ELSIF  parts.axes.statuses.initializationStatus.shutdown OR 
    parts.cover.statuses.initializationStatus.shutdown OR 
    parts.hydraulics.statuses.initializationStatus.shutdown OR 
    parts.m1.statuses.initializationStatus.shutdown OR 
    parts.m2.statuses.initializationStatus.shutdown OR 
    parts.m3.statuses.initializationStatus.shutdown OR 
    parts.safety.statuses.initializationStatus.shutdown OR 
    parts.services.statuses.initializationStatus.shutdown OR 
    parts.telemetry.statuses.initializationStatus.shutdown THEN

            statuses.initializationStatus(superState := TRUE, state := InitializationStates.SHUTDOWN);
ELSE
    statuses.initializationStatus(superState := FALSE);
END_IF


IF statuses.initializationStatus.initialized THEN
    IF statuses.healthStatus.bad THEN
        actualStatus := 'ERROR';
    ELSIF statuses.healthStatus.warning THEN
        actualStatus := 'Warning';
    ELSIF statuses.healthStatus.good THEN 
        IF statuses.busyStatus.busy THEN
            actualStatus := 'Busy';
        ELSIF statuses.busyStatus.idle THEN
            actualStatus := 'Idle';
        ELSE
            actualStatus := 'UNKNOWN';
        END_IF
    ELSE
        actualStatus := 'UNKNOWN';
	END_IF
ELSE
    actualStatus := InitializationStatusToString(statuses.initializationStatus);
END_IF


isInstrumentActive := parts.m3.statuses.busyStatus.idle AND parts.m3.actualKnownPositionID <> M3PositionIDs.UNKNOWN;

IF processes.changeInstrument.isBusy() THEN
    activeInstrumentName := 'Changing...';
    activeInstrumentNumber := -1;
ELSE
    IF isInstrumentActive THEN
        activeInstrumentName := parts.m3.actualKnownPositionName;
        
        IF activeInstrumentName = config.instruments.instrument0.name THEN
            activeInstrumentNumber := 0;
            activeInstrument := config.instruments.instrument0;
        ELSIF activeInstrumentName = config.instruments.instrument1.name THEN
            activeInstrumentNumber := 1;
            activeInstrument := config.instruments.instrument1;
        ELSIF activeInstrumentName = config.instruments.instrument2.name THEN
            activeInstrumentNumber := 2;
            activeInstrument := config.instruments.instrument2;
        ELSIF activeInstrumentName = config.instruments.instrument3.name THEN
            activeInstrumentNumber := 3;
            activeInstrument := config.instruments.instrument3;
        ELSIF activeInstrumentName = config.instruments.instrument4.name THEN
            activeInstrumentNumber := 4;
            activeInstrument := config.instruments.instrument4;
        ELSIF activeInstrumentName = config.instruments.instrument5.name THEN
            activeInstrumentNumber := 5;
            activeInstrument := config.instruments.instrument5;
        ELSIF activeInstrumentName = config.instruments.instrument6.name THEN
            activeInstrumentNumber := 6;
            activeInstrument := config.instruments.instrument6;
        ELSIF activeInstrumentName = config.instruments.instrument7.name THEN
            activeInstrumentNumber := 7;
            activeInstrument := config.instruments.instrument7;
        ELSIF activeInstrumentName = config.instruments.instrument8.name THEN
            activeInstrumentNumber := 8;
            activeInstrument := config.instruments.instrument8;
        ELSIF activeInstrumentName = config.instruments.instrument9.name THEN
            activeInstrumentNumber := 9;
            activeInstrument := config.instruments.instrument9;
        ELSE
            activeInstrumentNumber := -1;
		END_IF
            
    ELSE
        activeInstrumentName := 'None';
        activeInstrumentNumber := -1;
    END_IF
END_IF
END_METHOD

METHOD _shuttingDown
VAR_INPUT
END_VAR
IF processes.shutdown.statuses.busyStatus.busy THEN

    // make a rising edge for START:
	_nt_shutdown(START := FALSE);
	_nt_shutdown(NETID := '', 
               START := TRUE,
               DELAY := 0);

	// done
	processes.shutdown.setGood();
	processes.shutdown.setFinished();
END_IF
END_METHOD

METHOD _wakingUp
VAR_INPUT
END_VAR
IF processes.wakeUp.statuses.busyStatus.busy THEN
	
    CASE _wakeUpState OF
        0:
            parts.hydraulics.processes.startUpPumps.start();
            _wakeUpState := 1;
        1:
            IF parts.hydraulics.processes.startUpPumps.statuses.busyStatus.idle THEN
                IF parts.hydraulics.processes.startUpPumps.statuses.healthStatus.good THEN
                    _wakeUpState := 2;
                ELSE
                    _wakeUpState := 999;
                END_IF
			END_IF
        2:
            parts.axes.processes.powerOn.start(azi := TRUE, ele := TRUE, roc := FALSE, ron := FALSE, fw := FALSE);
            _wakeUpState := 3;
        3:
            IF isInstrumentActive THEN
                processes.changeInstrument.start(name := activeInstrumentName);
            END_IF
            _wakeUpState := 1000;
        999:
            // done with error
            processes.wakeUp.setBad();
            processes.wakeUp.setFinished();
            _wakeUpState := 0;
    
        1000:
            // done with error
            processes.wakeUp.setGood();
            processes.wakeUp.setFinished();
            _wakeUpState := 0;
    
	END_CASE


END_IF
END_METHOD

METHOD _changingInstrument 
VAR_INPUT
END_VAR
IF processes.changeInstrument.statuses.busyStatus.busy THEN
   
    CASE _changeInstrumentState OF
        
        0:
            processes.changeInstrument.setActualStatus('Changing...');
            
            // store the config of the given instrument
            IF processes.changeInstrument.get.name = config.instruments.instrument0.name THEN
                _changeInstrumentConfig := config.instruments.instrument0;
            ELSIF processes.changeInstrument.get.name = config.instruments.instrument1.name THEN
                _changeInstrumentConfig := config.instruments.instrument1;
            ELSIF processes.changeInstrument.get.name = config.instruments.instrument2.name THEN
                _changeInstrumentConfig := config.instruments.instrument2;
            ELSIF processes.changeInstrument.get.name = config.instruments.instrument3.name THEN
                _changeInstrumentConfig := config.instruments.instrument3;
            ELSIF processes.changeInstrument.get.name = config.instruments.instrument4.name THEN
                _changeInstrumentConfig := config.instruments.instrument4;
            ELSIF processes.changeInstrument.get.name = config.instruments.instrument5.name THEN
                _changeInstrumentConfig := config.instruments.instrument5;
            ELSIF processes.changeInstrument.get.name = config.instruments.instrument6.name THEN
                _changeInstrumentConfig := config.instruments.instrument6;
            ELSIF processes.changeInstrument.get.name = config.instruments.instrument7.name THEN
                _changeInstrumentConfig := config.instruments.instrument7;
            ELSIF processes.changeInstrument.get.name = config.instruments.instrument8.name THEN
                _changeInstrumentConfig := config.instruments.instrument8;
            ELSIF processes.changeInstrument.get.name = config.instruments.instrument9.name THEN
                _changeInstrumentConfig := config.instruments.instrument9;
            ELSE
                // wrong name
                _changeInstrumentState := 999;
			END_IF
            
            IF _changeInstrumentState <> 999 THEN
                _changeInstrumentState := 1;
			END_IF
            
        1:
            processes.changeInstrument.setActualStatus(CONCAT('Changing to ', _changeInstrumentConfig.name) );
            IF _changeInstrumentConfig.changeM3 THEN
                parts.m3.processes.gotoKnownPosition.start(name := _changeInstrumentConfig.name);
			END_IF
            IF _changeInstrumentConfig.doInitialThermalFocus THEN
                parts.m2.processes.doThermalFocusForStationName.start(station := _changeInstrumentConfig.name);
			END_IF
            IF _changeInstrumentConfig.moveKnownPosition THEN
                parts.axes.processes.moveKnownPosition.start(name := _changeInstrumentConfig.moveKnownPositionName);
			END_IF
            
            _changeInstrumentState := 2;
        2:
            IF       (parts.m3.processes.gotoKnownPosition.statuses.busyStatus.idle OR (NOT _changeInstrumentConfig.changeM3))
                AND  (parts.m2.processes.doThermalFocus.statuses.busyStatus.idle OR (NOT _changeInstrumentConfig.doInitialThermalFocus)) 
                AND  (parts.axes.processes.moveKnownPosition.statuses.busyStatus.idle OR (NOT _changeInstrumentConfig.moveKnownPosition))
            THEN
                IF       (parts.m3.processes.gotoKnownPosition.statuses.healthStatus.good OR (NOT _changeInstrumentConfig.changeM3))
                    AND  (parts.m2.processes.doThermalFocus.statuses.healthStatus.good OR (NOT _changeInstrumentConfig.doInitialThermalFocus))
                    AND  (parts.axes.processes.moveKnownPosition.statuses.healthStatus.good OR (NOT _changeInstrumentConfig.moveKnownPosition))
                THEN
                    _changeInstrumentState := 3;
                ELSIF parts.m3.processes.gotoKnownPosition.statuses.healthStatus.bad THEN
                    processes.changeInstrument.setActualStatus('M3 error');
                    _changeInstrumentState := 999;
                ELSIF parts.m2.processes.doThermalFocus.statuses.healthStatus.bad THEN
                    processes.changeInstrument.setActualStatus('M2 error');
                    _changeInstrumentState := 999;
                ELSIF parts.axes.processes.moveKnownPosition.statuses.healthStatus.bad THEN
                    processes.changeInstrument.setActualStatus('Axes error');
                    _changeInstrumentState := 999;
                ELSE
                    processes.changeInstrument.setActualStatus('ERROR'); // should not be happening
                    _changeInstrumentState := 999;
                END_IF
			END_IF
        3:
            // power off has priority over power on
            IF _changeInstrumentConfig.powerOffRoc THEN
                parts.axes.parts.roc.processes.powerOff.start();
                _changeInstrumentState := 4;
            ELSIF _changeInstrumentConfig.powerOnRoc THEN
                parts.axes.parts.roc.processes.powerOn.start();
                _changeInstrumentState := 5;
            ELSE
                _changeInstrumentState := 6;
			END_IF
        4:
            IF parts.axes.parts.roc.processes.powerOff.isIdle() THEN
                IF parts.axes.parts.roc.processes.powerOff.isGood() THEN
                    _changeInstrumentState := 6;
                ELSE
                    _changeInstrumentState := 999;
                    processes.changeInstrument.setActualStatus('ROC error');
				END_IF
			END_IF
        5:
            IF parts.axes.parts.roc.processes.powerOn.isIdle() THEN
                IF parts.axes.parts.roc.processes.powerOn.isGood() THEN
                    _changeInstrumentState := 6;
                ELSE
                    _changeInstrumentState := 999;
                    processes.changeInstrument.setActualStatus('ROC error');
				END_IF
			END_IF
        6:
            // power off has priority over power on
            IF _changeInstrumentConfig.powerOffRon THEN
                parts.axes.parts.ron.processes.powerOff.start();
                _changeInstrumentState := 7;
            ELSIF _changeInstrumentConfig.powerOnRon THEN
                parts.axes.parts.ron.processes.powerOn.start();
                _changeInstrumentState := 8;
            ELSE
                _changeInstrumentState := 9;
			END_IF
        7:
            IF parts.axes.parts.ron.processes.powerOff.isIdle() THEN
                IF parts.axes.parts.ron.processes.powerOff.isGood() THEN
                    _changeInstrumentState := 9;
                ELSE
                    _changeInstrumentState := 999;
                    processes.changeInstrument.setActualStatus('RON error');
				END_IF
			END_IF
        8:
            IF parts.axes.parts.ron.processes.powerOn.isIdle() THEN
                IF parts.axes.parts.ron.processes.powerOn.isGood() THEN
                    _changeInstrumentState := 9;
                ELSE
                    _changeInstrumentState := 999;
                    processes.changeInstrument.setActualStatus('RON error');
				END_IF
			END_IF
        9:
            IF _changeInstrumentConfig.loadPointingModel THEN
                parts.axes.processes.enablePointingModel.start(name := _changeInstrumentConfig.name);
                _changeInstrumentState := 10;
            ELSE
                _changeInstrumentState := 11;
			END_IF
        10:
            IF parts.axes.processes.enablePointingModel.isIdle() THEN
                IF parts.axes.processes.enablePointingModel.isGood() THEN
                    _changeInstrumentState := 11;
                ELSE
                    _changeInstrumentState := 999;
                    processes.changeInstrument.setActualStatus('TPOINT error');
				END_IF
			END_IF
        11:
            // done (rotator active/inactive is automatically updated by axes)
            _changeInstrumentState := 1000;
            processes.changeInstrument.setActualStatus(CONCAT('Changed to ', _changeInstrumentConfig.name));
        999:
            // done with error
            processes.changeInstrument.setBad();
            processes.changeInstrument.setFinished();
            _changeInstrumentState := 0;
    
        1000:
            // done with error
            processes.changeInstrument.setGood();
            processes.changeInstrument.setFinished();
            _changeInstrumentState := 0;
	END_CASE
    
END_IF
END_METHOD

METHOD _changingOperator 
VAR_INPUT
END_VAR
IF processes.changeOperator.statuses.busyStatus.busy THEN
    // ok we're started
	processes.changeOperator.setStarted();
    
    // depending on the state, we'll check the password (or not)
    IF processes.changeOperator.get.state = OperatorStates.TECH THEN
        // check the password for TECH!    
        IF processes.changeOperator.get.password = GLOBAL.config.PASSWORD_TECH THEN
            // ok!
            noOfFailedOperatorChanges := 0;
            statuses.operatorStatus(state := OperatorStates.TECH);
            processes.changeOperator.setGood();
            processes.changeOperator.setFinished();
        ELSE
            // wrong password!
            noOfFailedOperatorChanges := noOfFailedOperatorChanges + 1;
            processes.changeOperator.setBad();
            processes.changeOperator.setFinished();
		END_IF
    ELSE
        // no password needed
        statuses.operatorStatus(state := processes.changeOperator.get.state);
        processes.changeOperator.setGood();
	    processes.changeOperator.setFinished();
	END_IF
    
    // whether or not we logged in, there needs to be a new password entered,
    // so the current status is again 'bad'!
    statuses.passwordHealthStatus(isGood := FALSE);
END_IF
END_METHOD

METHOD FB_init : BOOL
VAR_INPUT
	bInitRetains : BOOL; // if TRUE, the retain variables are initialized (warm start / cold start)
	bInCopyCode : BOOL;  // if TRUE, the instance afterwards gets moved into the copy code (online change)
END_VAR
processes.changeOperator.start(state := OperatorStates.OBSERVER, password := '');

parts.configManager.configure(
    editableConfigAddress       := ADR(editableConfig),
    activeConfigAddress         := ADR(config),
    configLength                := SIZEOF(editableConfig),
    editableConfigSymbolName    := GLOBAL.config.MTCS_EDITABLE_CONFIG_SYMBOL_NAME,
    activeConfigSymbolName      := GLOBAL.config.MTCS_ACTIVE_CONFIG_SYMBOL_NAME,
    configFilePath              := GLOBAL.config.MTCS_CONFIG_FILE_PATH);
END_METHOD

METHOD _goingToSleep
VAR_INPUT
END_VAR
IF processes.goToSleep.statuses.busyStatus.busy THEN
    
    CASE _goToSleepState OF
        0:
            parts.axes.processes.powerOff.start();
            _goToSleepState := 1;
        1:
            IF parts.axes.processes.powerOff.statuses.busyStatus.idle THEN
                // regardless of success or failure, go to the next step
                _goToSleepState := 2;
			END_IF
        2:
            parts.hydraulics.processes.stopPumps.start();
            _goToSleepState := 3;
        3:
            IF parts.hydraulics.processes.stopPumps.statuses.busyStatus.idle THEN
                IF parts.hydraulics.processes.stopPumps.statuses.healthStatus.good THEN
                    _goToSleepState := 1000;
                ELSE
                    _goToSleepState := 999;
                END_IF
			END_IF
        999:
            // done with error
            processes.goToSleep.setBad();
            processes.goToSleep.setFinished();
            _goToSleepState := 0;
    
        1000:
            // done with error
            processes.goToSleep.setGood();
            processes.goToSleep.setFinished();
            _goToSleepState := 0;
    
	END_CASE


END_IF
END_METHOD

METHOD _rebooting
VAR_INPUT
END_VAR
IF processes.reboot.statuses.busyStatus.busy THEN

    // make a rising edge for START:
	_nt_reboot(START := FALSE);
	_nt_reboot(NETID := '', 
               START := TRUE,
               DELAY := 0);

	// done
	processes.reboot.setGood();
	processes.reboot.setFinished();
END_IF
END_METHOD

METHOD _locking
VAR_INPUT
END_VAR
IF processes.lock.statuses.busyStatus.busy THEN
	statuses.initializationStatus(state := InitializationStates.LOCKED);
	
	// done
	processes.lock.setGood();
	processes.lock.setFinished();
END_IF
END_METHOD

METHOD _verifyingPassword 
VAR_INPUT
END_VAR
IF processes.verifyPassword.isBusy() THEN
    // ok we're started
	processes.verifyPassword.setStarted();
    
    // depending on the state, we'll check the password (or not)
    IF processes.verifyPassword.get.state = OperatorStates.TECH THEN
        // check the password for TECH!    
        IF processes.verifyPassword.get.password = GLOBAL.config.PASSWORD_TECH THEN
            // ok!
            noOfFailedOperatorChanges := 0;
            statuses.passwordHealthStatus(isGood := TRUE);
            processes.verifyPassword.setGood();
            processes.verifyPassword.setFinished();
        ELSE
            // wrong password!
            noOfFailedOperatorChanges := noOfFailedOperatorChanges + 1;
            statuses.passwordHealthStatus(isGood := FALSE);
            processes.verifyPassword.setBad();
            processes.verifyPassword.setFinished();
		END_IF
    ELSE
        // no password needed
        statuses.operatorStatus(state := processes.changeOperator.get.state);
        // there was no password needed, so we can "reset" the password health status again:
        statuses.passwordHealthStatus(isGood := FALSE);
        processes.changeOperator.setGood();
	    processes.changeOperator.setFinished();
	END_IF
END_IF
END_METHOD

METHOD _unlocking
VAR_INPUT
END_VAR
IF processes.unlock.statuses.busyStatus.busy THEN
	statuses.initializationStatus(state := InitializationStates.INITIALIZED);
	
	// done
	processes.unlock.setGood();
	processes.unlock.setFinished();
END_IF
END_METHOD

METHOD _initializing
VAR_INPUT
END_VAR
VAR
    
END_VAR
IF processes.initialize.statuses.busyStatus.busy THEN
	
	// start up the initialization
	IF NOT processes.initialize.statuses.startedStatus.started THEN
        // we're now initializing
        _initializingCurrentAction := 0;
		// OK we're started now
		processes.initialize.setStarted();
	END_IF;
    
    // process the actions
    CASE _initializingCurrentAction OF
        0:
            // first initialize the safety
            parts.safety.processes.initialize.start();
            _initializingCurrentAction := 1;
        1:
            // wait until the safety is initialized
            IF parts.safety.processes.initialize.isIdle() THEN
                _initializingCurrentAction := 2;
			END_IF
        2:
            // start initializing everything
            parts.cover.processes.initialize.start();
            parts.m1.processes.initialize.start();
            parts.m2.processes.initialize.start();
            parts.m3.processes.initialize.start();
            parts.services.processes.initialize.start();
            parts.telemetry.processes.initialize.start();
            parts.hydraulics.processes.initialize.start();
            _initializingCurrentAction := 3;
        3:
            // wait until everything is initialized
            IF     parts.cover.processes.initialize.isIdle() 
               AND parts.m1.processes.initialize.isIdle() 
               AND parts.m3.processes.initialize.isIdle() 
               AND parts.m2.processes.initialize.isIdle() 
               AND parts.services.processes.initialize.isIdle() 
               AND parts.telemetry.processes.initialize.isIdle() 
               AND parts.hydraulics.processes.initialize.isIdle() 
            THEN
                IF     parts.cover.processes.initialize.isGood() 
                   AND parts.m1.processes.initialize.isGood() 
                   AND parts.m2.processes.initialize.isGood() 
                   AND parts.m3.processes.initialize.isGood() 
                   AND parts.services.processes.initialize.isGood() 
                   AND parts.telemetry.processes.initialize.isGood() 
                   AND parts.hydraulics.processes.initialize.isGood() 
                THEN
                    _initializingCurrentAction := 4;
                ELSE
                    _initializingCurrentAction := 999;
                END_IF
            END_IF
        4:
            parts.hydraulics.processes.startUpPumps.start();
            _initializingCurrentAction := 5;
        5:
            IF parts.hydraulics.processes.startUpPumps.isIdle() THEN
                IF parts.hydraulics.processes.startUpPumps.isGood() THEN
                    _initializingCurrentAction := 6;
                ELSE
                    _initializingCurrentAction := 999;
                END_IF
			END_IF
        6:
            parts.axes.processes.initialize.start();
            _initializingCurrentAction := 7;
        7:
            IF parts.axes.processes.initialize.isIdle() THEN
                IF parts.axes.processes.initialize.isGood() THEN
                    _initializingCurrentAction := 8;
                ELSE
                    _initializingCurrentAction := 999;
				END_IF
            END_IF
        8:
            IF isInstrumentActive THEN
                processes.changeInstrument.start(name := activeInstrumentName);
            END_IF
            _initializingCurrentAction := 1000;
        999:
            // there has been an error!
            // done
            processes.initialize.setBad();
            processes.initialize.setFinished();
        1000:
            // all done!
            processes.initialize.setGood();
            processes.initialize.setFinished();
	END_CASE
    
END_IF
END_METHOD

END_FUNCTION_BLOCK

// ---- MTCS/Common/StateMachines/ConfigManager.TcPOU
FUNCTION_BLOCK ConfigManager EXTENDS SM_ConfigManager
VAR_INPUT
END_VAR
VAR_OUTPUT
END_VAR
VAR;
    xmlRead : FB_XmlSrvReadByName;
    xmlWrite : FB_XmlSrvWriteByName;
    
    _editableConfigAddress : PVOID := 0;
    _activeConfigAddress : PVOID := 0;
    _configLength : UDINT;
    _editableConfigSymbolName : STRING;
    _activeConfigSymbolName : STRING;
    _configFilePath : STRING;
END_VAR

SUPER^();

_loading();
_saving();
_activating();

SUPER^();

METHOD _activating : BOOL
VAR_INPUT
END_VAR
IF processes.activate.statuses.busyStatus.busy THEN
    
    IF _editableConfigAddress <> 0 AND _activeConfigAddress <> 0 AND _configLength > 0 THEN
        MEMCPY(_activeConfigAddress, _editableConfigAddress, _configLength);
        processes.activate.setGood();
    ELSE
        processes.activate.setBad();
	END_IF
    
    processes.activate.setFinished();

END_IF
END_METHOD

METHOD configure
VAR_INPUT
    editableConfigAddress : PVOID := 0;
    activeConfigAddress : PVOID := 0;
    configLength : UDINT;
    editableConfigSymbolName : STRING;
    activeConfigSymbolName : STRING;
    configFilePath : STRING;
END_VAR
_editableConfigAddress := editableConfigAddress;
_activeConfigAddress := activeConfigAddress;
_configLength := configLength;
_editableConfigSymbolName := editableConfigSymbolName;
_activeConfigSymbolName := activeConfigSymbolName;
_configFilePath := configFilePath;
END_METHOD

METHOD _saving : BOOL
VAR_INPUT
END_VAR
IF processes.save.statuses.busyStatus.busy THEN
	
    // write the file to the local directory
    xmlWrite(
        sNetId := '',
        nMode := XMLSRV_ADDMISSING,
        sSymName := _activeConfigSymbolName,
        sFilePath := _configFilePath,
        sXPath := '/config',
        bExecute := TRUE,
        tTimeout := T#10S);
        
	(* update the busy status *)
	processes.save.statuses.busyStatus(isBusy := xmlWrite.bBusy);
	
	(* update the health status *)
	processes.save.statuses.healthStatus(isGood := NOT xmlWrite.bError);
    
    (* update the error ID *)
    processes.save.errorId := xmlWrite.nErrId;
    
    IF NOT xmlWrite.bBusy THEN
        // reset the trigger
        xmlWrite(bExecute := FALSE);
    END_IF
    
END_IF
END_METHOD

METHOD _loading : BOOL
VAR_INPUT
END_VAR
IF processes.load.statuses.busyStatus.busy THEN
	
    IF NOT processes.load.statuses.startedStatus.started THEN
        // read the file
        xmlRead(
            sNetId := '',
            nMode := XMLSRV_SKIPMISSING,
            sSymName := _editableConfigSymbolName,
            sFilePath := _configFilePath,
            sXPath := 'config',
            bExecute := TRUE,
            tTimeout := T#5S);
        
        processes.load.setStarted();
    ELSE
        xmlRead(bExecute := FALSE);
	END_IF
    
	(* update the busy status *)
	processes.load.statuses.busyStatus(isBusy := xmlRead.bBusy);
	
	(* update the health status *)
	processes.load.statuses.healthStatus(isGood := NOT xmlRead.bError);
    
    (* update the error ID *)
    processes.load.errorId := xmlRead.nErrId;
    
END_IF
END_METHOD

END_FUNCTION_BLOCK

// ---- MTCS/Axes/StateMachines/Axes.TcPOU
FUNCTION_BLOCK Axes EXTENDS SM_Axes
VAR_INPUT
    
END_VAR
VAR_OUTPUT
END_VAR
VAR
    _onFirstStartCurrentAction : INT;
    
	doPointingTon : TON;
	_relativePointingTon : TON;
	_relativePointOldAz: LREAL;
	_relativePointOldEl: LREAL;
    
    _relativePointDeltaAzi : LREAL;
    _relativePointDeltaEle : LREAL;
    
    _errorMonitoringTon : TON;
    _slipMonitoringEdgeDetection : R_TRIG;
    _personHasEnteredMonitoringEdgeDetection : R_TRIG;
    
    _aziStoMonitoringEdgeDetection : F_TRIG;
    _eleStoMonitoringEdgeDetection : F_TRIG;
    _rocStoMonitoringEdgeDetection : F_TRIG;
    _ronStoMonitoringEdgeDetection : F_TRIG;
    
    _limitsReachedEdgeDetection : R_TRIG;
    
    _aziStoCounter : INT;
    _eleStoCounter : INT;
    _rocStoCounter : INT;
    _ronStoCounter : INT;
    
	_trackingStartAzi : LREAL;  // degrees!
	_trackingStartEle : LREAL;  // degrees!
	_trackingStartRot : LREAL;  // degrees!
    
    _tpointCalculations : AxesTPointCalculations;
    _tpointFeedbackCalculations : AxesTPointCalculations;
    
    _aziPointingMoveCalculator : AxesMoveAbsoluteCalculator;
    _elePointingMoveCalculator : AxesMoveAbsoluteCalculator;
    _rocPointingMoveCalculator : AxesMoveAbsoluteCalculator;
    _ronPointingMoveCalculator : AxesMoveAbsoluteCalculator;
    
    _pointRocRequested : BOOL;
    _pointRonRequested : BOOL;
    _pointRocOffset : LREAL;
    _pointRonOffset : LREAL;
    
    _aziMoveRelativeCalculator : AxesMoveRelativeCalculator;
    _eleMoveRelativeCalculator : AxesMoveRelativeCalculator;
    _rocMoveRelativeCalculator : AxesMoveRelativeCalculator;
    _ronMoveRelativeCalculator : AxesMoveRelativeCalculator;
    
	_alphaVelocityStartTimeS: LREAL; // seconds
    
	{attribute 'OPC.UA.DA' := '0'}
    _slalibSmoothener : AxesSlalibSmoothener;
    
	{attribute 'OPC.UA.DA' := '0'}
    _actualKnownPositionConfig : AxesKnownPositionConfig;
    
    _setTargetTon : TON;
    
    
    _isPoweredOffByPersonInDome_azi : BOOL;
    _isPoweredOffByPersonInDome_ele : BOOL;
    _isPoweredOffByPersonInDome_roc : BOOL;
    _isPoweredOffByPersonInDome_ron : BOOL;
END_VAR

_update();


_onFirstStart();
_initializing();
_resetting();
_changingOperatingState();
_locking();
_unlocking();
_setAlphaDeltaVelocity();
_applyAlphaDeltaVelocity();

_enablePointingModel();
_disablePointingModel();

_doHoming();
_setTarget();
_point();
_powerOn();
_powerOff();
_moveAbsolute();
_moveRelative();
_stop();
_quickStop();

// call the _callOnce method, which contains logic
// that may only be called once per task cycle!
_callOnce();

_pointRelative();

_slipMonitoring();
_errorMonitoring();
_stoMonitoring();
_limitMonitoring();
_domeAccessMonitoring();
_moveKnownPosition();

_update();

METHOD _limitMonitoring
VAR_INPUT
END_VAR
_limitsReachedEdgeDetection(CLK :=    
       (parts.azi.statuses.poweredStatus.enabled AND parts.azi.setPosLimitReached)
    OR (parts.ele.statuses.poweredStatus.enabled AND parts.ele.setPosLimitReached)
    OR (parts.roc.statuses.poweredStatus.enabled AND parts.roc.setPosLimitReached)
    OR (parts.ron.statuses.poweredStatus.enabled AND parts.ron.setPosLimitReached));
    
IF _limitsReachedEdgeDetection.Q THEN
    isLimitsReached := TRUE;
    processes.stop.start();
END_IF


// reset the isLimitsFlag with the following commands:
IF     processes.point.isBusy() 
    OR processes.doHoming.isBusy()
    OR processes.moveAbsolute.isBusy()
    OR processes.moveKnownPosition.isBusy()
    OR processes.powerOff.isBusy()
    OR processes.powerOn.isBusy()
    OR processes.reset.isBusy() THEN
    isLimitsReached := FALSE;
END_IF
END_METHOD

METHOD _powerOff
VAR_INPUT
END_VAR
IF processes.powerOff.isBusy() THEN
    
    IF NOT processes.powerOff.isStarted() THEN
        processes.powerOff.state := 0;
        processes.powerOff.setStarted();
	END_IF
    
    CASE processes.powerOff.state OF
        0:
            processes.powerOff.setActualStatus('Powering off the axes');
            // now power off the axes
            parts.azi.processes.powerOff.start();
            parts.ele.processes.powerOff.start();
            parts.roc.processes.powerOff.start();
            parts.ron.processes.powerOff.start();
            processes.powerOff.state := 1;
        1:
            IF      parts.azi.processes.powerOff.isIdle() 
                AND parts.ele.processes.powerOff.isIdle()  
                AND parts.roc.processes.powerOff.isIdle()  
                AND parts.ron.processes.powerOff.isIdle() THEN
                
                IF      parts.azi.processes.powerOff.isGood() 
                   AND  parts.ele.processes.powerOff.isGood() 
                   AND  parts.roc.processes.powerOff.isGood() 
                   AND  parts.ron.processes.powerOff.isGood() THEN
                    // ok, all axes are powered off
                    processes.powerOff.state := 1000;
                ELSE
                    processes.powerOff.setActualStatus('Could not power off the axes!');
                    processes.powerOff.state := 999;
                END_IF
            END_IF
        999:
            // error!
            processes.powerOff.setBad();
            processes.powerOff.setFinished();
            // stop all axes
            processes.stop.start();
        1000:
            processes.powerOff.setActualStatus('Powered off');
            // ok done
            processes.powerOff.setFinished();
            processes.powerOff.setGood();
		
    END_CASE
    
END_IF
END_METHOD

METHOD _enablePointingModel
VAR_INPUT
END_VAR
IF processes.enablePointingModel.isBusy() THEN
    
    IF processes.enablePointingModel.get.name = '' THEN
        processes.enablePointingModel.setActualStatus('Invalid model name');
    ELSIF processes.enablePointingModel.get.name = parts.tpoint.parts.model0.config.name THEN
        activePointingModel := parts.tpoint.parts.model0.config;
        activePointingModelNumber := 0;
        isPointingModelActive := TRUE;
    ELSIF processes.enablePointingModel.get.name = parts.tpoint.parts.model1.config.name THEN
        activePointingModel := parts.tpoint.parts.model1.config;
        activePointingModelNumber := 1;
        isPointingModelActive := TRUE;
    ELSIF processes.enablePointingModel.get.name = parts.tpoint.parts.model2.config.name THEN
        activePointingModel := parts.tpoint.parts.model2.config;
        activePointingModelNumber := 2;
        isPointingModelActive := TRUE;
    ELSIF processes.enablePointingModel.get.name = parts.tpoint.parts.model3.config.name THEN
        activePointingModel := parts.tpoint.parts.model3.config;
        activePointingModelNumber := 3;
        isPointingModelActive := TRUE;
    ELSIF processes.enablePointingModel.get.name = parts.tpoint.parts.model4.config.name THEN
        activePointingModel := parts.tpoint.parts.model4.config;
        activePointingModelNumber := 4;
        isPointingModelActive := TRUE;
    ELSIF processes.enablePointingModel.get.name = parts.tpoint.parts.model5.config.name THEN
        activePointingModel := parts.tpoint.parts.model5.config;
        activePointingModelNumber := 5;
        isPointingModelActive := TRUE;
    ELSIF processes.enablePointingModel.get.name = parts.tpoint.parts.model6.config.name THEN
        activePointingModel := parts.tpoint.parts.model6.config;
        activePointingModelNumber := 6;
        isPointingModelActive := TRUE;
    ELSIF processes.enablePointingModel.get.name = parts.tpoint.parts.model7.config.name THEN
        activePointingModel := parts.tpoint.parts.model7.config;
        activePointingModelNumber := 7;
        isPointingModelActive := TRUE;
    ELSIF processes.enablePointingModel.get.name = parts.tpoint.parts.model8.config.name THEN
        activePointingModel := parts.tpoint.parts.model8.config;
        activePointingModelNumber := 8;
        isPointingModelActive := TRUE;
    ELSIF processes.enablePointingModel.get.name = parts.tpoint.parts.model9.config.name THEN
        activePointingModel := parts.tpoint.parts.model9.config;
        activePointingModelNumber := 9;
        isPointingModelActive := TRUE;
    ELSE
        processes.enablePointingModel.setActualStatus(CONCAT('Model ', CONCAT( processes.enablePointingModel.get.name, '$' not found')));
	END_IF

    IF isPointingModelActive THEN
        processes.enablePointingModel.setActualStatus(CONCAT('Loaded model ', CONCAT( processes.enablePointingModel.get.name, '$'')));
        processes.enablePointingModel.setGood();
    ELSE
        processes.enablePointingModel.setBad();
	END_IF
    
    _update_activePointingModel();
    
    
    processes.enablePointingModel.setFinished();
    
END_IF
END_METHOD

METHOD _disablePointingModel
VAR_INPUT
END_VAR
IF processes.disablePointingModel.isBusy() THEN
    
    isPointingModelActive := FALSE;
    activePointingModelNumber := -1;
    processes.disablePointingModel.setActualStatus('No model loaded');
    processes.disablePointingModel.setGood();
    processes.disablePointingModel.setFinished();
    
END_IF
END_METHOD

METHOD _setAlphaDeltaVelocity
VAR_INPUT
END_VAR
VAR
    alphaVeloDegPerSec : LREAL;
    deltaVeloDegPerSec : LREAL;
    alphaVeloArcsecPerSec : LREAL;
    deltaVeloArcsecPerSec : LREAL;
    alphaVeloArcsecPerHour : LREAL;
    deltaVeloArcsecPerHour : LREAL;
    msg : STRING;
    _formatStr : FB_FormatString;
END_VAR
IF processes.setAlphaDeltaVelocity.isBusy() THEN

    alphaVeloDegPerSec := AxesMoveVelocityUnitsToDegPerSec(units := processes.setAlphaDeltaVelocity.get.units, value := processes.setAlphaDeltaVelocity.get.alphaVelocity);
    deltaVeloDegPerSec := AxesMoveVelocityUnitsToDegPerSec(units := processes.setAlphaDeltaVelocity.get.units, value := processes.setAlphaDeltaVelocity.get.deltaVelocity);
    
    target.alphaVelocity(newDegreesPerSecondValue := alphaVeloDegPerSec);
    target.deltaVelocity(newDegreesPerSecondValue := deltaVeloDegPerSec);
    
    _alphaVelocityStartTimeS := GLOBAL.config.TIME_NOW_S;
    
    alphaVeloArcsecPerSec := DEG_TO_ARCSEC(alphaVeloDegPerSec);
    deltaVeloArcsecPerSec := DEG_TO_ARCSEC(deltaVeloDegPerSec);
    
    IF ABS(alphaVeloArcsecPerSec) < 0.0000000001 AND ABS(deltaVeloArcsecPerSec) < 0.0000000001 THEN
        msg := 'Stopped';
    ELSIF ABS(alphaVeloArcsecPerSec) < 0.005 OR ABS(deltaVeloArcsecPerSec) < 0.005 THEN 
        alphaVeloArcsecPerHour := alphaVeloArcsecPerSec * 3600.0;
        deltaVeloArcsecPerHour := deltaVeloArcsecPerSec * 3600.0;
        _formatStr(
            sFormat := 'Move alpha=%.3f"/h delta=%.3f"/h', 
            arg1 := F_LREAL(alphaVeloArcsecPerHour),
            arg2 := F_LREAL(alphaVeloArcsecPerHour), 
            sOut => msg);
    ELSIF alphaVeloArcsecPerSec < 0.1 OR deltaVeloArcsecPerSec < 0.1 THEN 
        _formatStr(
            sFormat := 'Move alpha=%.5f"/s delta=%.5f"/s', 
            arg1 := F_LREAL(alphaVeloArcsecPerSec),
            arg2 := F_LREAL(deltaVeloArcsecPerSec), 
            sOut => msg);
    ELSE
        _formatStr(
            sFormat := 'Move alpha=%.3f"/s delta=%.3f"/s', 
            arg1 := F_LREAL(alphaVeloArcsecPerSec),
            arg2 := F_LREAL(deltaVeloArcsecPerSec), 
            sOut => msg);
	END_IF
    
    
    processes.setAlphaDeltaVelocity.setActualStatus(msg);
    processes.setAlphaDeltaVelocity.setGood();
    processes.setAlphaDeltaVelocity.setFinished();
    
END_IF
END_METHOD

METHOD _applyAlphaDeltaVelocity
VAR_INPUT
END_VAR
VAR
END_VAR

IF target.alphaVelocity.degreesPerSecond.value <> 0 THEN
    target.alphaTravelled(newDegreesValue := target.alphaTravelled.degrees.value + TIME_TO_LREAL(GLOBAL.config.PLC_FAST_TASK_TIME) / 1000.0 * target.alphaVelocity.degreesPerSecond.value);    
END_IF
IF target.deltaVelocity.degreesPerSecond.value <> 0 THEN
    target.deltaTravelled(newDegreesValue := target.deltaTravelled.degrees.value + TIME_TO_LREAL(GLOBAL.config.PLC_FAST_TASK_TIME) / 1000.0 * target.deltaVelocity.degreesPerSecond.value);    
END_IF
END_METHOD

METHOD _resetting
VAR_INPUT
END_VAR
VAR
    
END_VAR
IF processes.reset.statuses.busyStatus.busy THEN
	
	// start up the initialization
	IF NOT processes.reset.statuses.startedStatus.started THEN
        processes.reset._state := 0;
		// OK we're started now
		processes.reset.setStarted();
	END_IF;
    
    // process the actions
    CASE processes.reset._state OF
        
        0:
            // reset all processes so that they are green again
            processes.changeOperatingState.resetIfIdle();
            processes.disablePointingModel.resetIfIdle();
            processes.doHoming.resetIfIdle();
            processes.enablePointingModel.resetIfIdle();
            processes.lock.resetIfIdle();
            processes.initialize.resetIfIdle();
            processes.moveAbsolute.resetIfIdle();
            processes.moveKnownPosition.resetIfIdle();
            processes.moveRelative.resetIfIdle();
            processes.point.resetIfIdle();
            processes.pointRelative.resetIfIdle();
            processes.powerOff.resetIfIdle();
            processes.powerOn.resetIfIdle();
            processes.quickStop.resetIfIdle();
            processes.setAlphaDeltaVelocity.resetIfIdle();
            processes.setTarget.resetIfIdle();
            processes.stop.resetIfIdle();
            processes.unlock.resetIfIdle();
            
            processes.reset.setActualStatus('Loading the configs from XML files');
            parts.configManager.processes.load.start(parts.configManager.processes.load.set.filePath);
            processes.reset._state := 1;
        1:
            IF parts.configManager.processes.load.statuses.busyStatus.idle THEN
                IF parts.configManager.processes.load.statuses.healthStatus.good THEN
                    processes.reset._state := 2;
                ELSE
                    processes.reset.setActualStatus('Failed to load the config');
                    processes.reset._state := 999;
                END_IF
            END_IF
        2:
            processes.reset.setActualStatus('Activating the config');
            parts.configManager.processes.activate.start();
            processes.reset._state := 3;
        3:
            // wait until the config has been activated
            IF parts.configManager.processes.activate.statuses.busyStatus.idle THEN
                IF parts.configManager.processes.activate.statuses.healthStatus.good THEN
                    processes.reset._state := 4;
                ELSE
                    processes.reset.setActualStatus('Failed to activate the config');
                    processes.reset._state := 999;
                END_IF
            END_IF
        4:
            // start loading the TPoint models from XML file
            parts.tpoint.parts.model0.parts.configManager.processes.load.start(parts.tpoint.parts.model0.parts.configManager.processes.load.set.filePath);
            parts.tpoint.parts.model1.parts.configManager.processes.load.start(parts.tpoint.parts.model1.parts.configManager.processes.load.set.filePath);
            parts.tpoint.parts.model2.parts.configManager.processes.load.start(parts.tpoint.parts.model2.parts.configManager.processes.load.set.filePath);
            parts.tpoint.parts.model3.parts.configManager.processes.load.start(parts.tpoint.parts.model3.parts.configManager.processes.load.set.filePath);
            parts.tpoint.parts.model4.parts.configManager.processes.load.start(parts.tpoint.parts.model4.parts.configManager.processes.load.set.filePath);
            parts.tpoint.parts.model5.parts.configManager.processes.load.start(parts.tpoint.parts.model5.parts.configManager.processes.load.set.filePath);
            parts.tpoint.parts.model6.parts.configManager.processes.load.start(parts.tpoint.parts.model6.parts.configManager.processes.load.set.filePath);
            parts.tpoint.parts.model7.parts.configManager.processes.load.start(parts.tpoint.parts.model7.parts.configManager.processes.load.set.filePath);
            parts.tpoint.parts.model8.parts.configManager.processes.load.start(parts.tpoint.parts.model8.parts.configManager.processes.load.set.filePath);
            parts.tpoint.parts.model9.parts.configManager.processes.load.start(parts.tpoint.parts.model9.parts.configManager.processes.load.set.filePath);
            processes.reset._state := 5;
        5:
            // wait until the configs have been loaded
            IF     parts.tpoint.parts.model0.parts.configManager.processes.load.statuses.busyStatus.idle
               AND parts.tpoint.parts.model1.parts.configManager.processes.load.statuses.busyStatus.idle 
               AND parts.tpoint.parts.model2.parts.configManager.processes.load.statuses.busyStatus.idle 
               AND parts.tpoint.parts.model3.parts.configManager.processes.load.statuses.busyStatus.idle 
               AND parts.tpoint.parts.model4.parts.configManager.processes.load.statuses.busyStatus.idle 
               AND parts.tpoint.parts.model5.parts.configManager.processes.load.statuses.busyStatus.idle 
               AND parts.tpoint.parts.model6.parts.configManager.processes.load.statuses.busyStatus.idle 
               AND parts.tpoint.parts.model7.parts.configManager.processes.load.statuses.busyStatus.idle 
               AND parts.tpoint.parts.model8.parts.configManager.processes.load.statuses.busyStatus.idle 
               AND parts.tpoint.parts.model9.parts.configManager.processes.load.statuses.busyStatus.idle 
            THEN
                // some files may have failed to load, because not all models may be present
                processes.reset._state := 6;
            END_IF
        6:
            // now start activating the configs
            parts.tpoint.parts.model0.parts.configManager.processes.activate.start();
            parts.tpoint.parts.model1.parts.configManager.processes.activate.start();
            parts.tpoint.parts.model2.parts.configManager.processes.activate.start();
            parts.tpoint.parts.model3.parts.configManager.processes.activate.start();
            parts.tpoint.parts.model4.parts.configManager.processes.activate.start();
            parts.tpoint.parts.model5.parts.configManager.processes.activate.start();
            parts.tpoint.parts.model6.parts.configManager.processes.activate.start();
            parts.tpoint.parts.model7.parts.configManager.processes.activate.start();
            parts.tpoint.parts.model8.parts.configManager.processes.activate.start();
            parts.tpoint.parts.model9.parts.configManager.processes.activate.start();
            processes.reset._state := 7;
        7:
            // wait until the configs have been activated
            IF      parts.tpoint.parts.model0.parts.configManager.processes.activate.statuses.busyStatus.idle 
                AND parts.tpoint.parts.model1.parts.configManager.processes.activate.statuses.busyStatus.idle 
                AND parts.tpoint.parts.model2.parts.configManager.processes.activate.statuses.busyStatus.idle 
                AND parts.tpoint.parts.model3.parts.configManager.processes.activate.statuses.busyStatus.idle 
                AND parts.tpoint.parts.model4.parts.configManager.processes.activate.statuses.busyStatus.idle 
                AND parts.tpoint.parts.model5.parts.configManager.processes.activate.statuses.busyStatus.idle 
                AND parts.tpoint.parts.model6.parts.configManager.processes.activate.statuses.busyStatus.idle 
                AND parts.tpoint.parts.model7.parts.configManager.processes.activate.statuses.busyStatus.idle 
                AND parts.tpoint.parts.model8.parts.configManager.processes.activate.statuses.busyStatus.idle 
                AND parts.tpoint.parts.model9.parts.configManager.processes.activate.statuses.busyStatus.idle 
            THEN
                processes.reset._state := 8;
            END_IF
        8:
            processes.reset.setActualStatus('Resetting the axes');
            parts.azi.processes.reset.start();
            parts.ele.processes.reset.start();
            parts.roc.processes.reset.start();
            parts.ron.processes.reset.start();
            processes.reset._state := 9;
            //parts.fwAxis.processes.reset.start();TODO!!
        9:
            IF      parts.azi.processes.reset.isIdle() 
                AND parts.ele.processes.reset.isIdle() 
                AND parts.roc.processes.reset.isIdle() 
                AND parts.ron.processes.reset.isIdle() 
                // parts.fwAxis.processes.reset.start()
            THEN
                IF      parts.azi.processes.reset.isGood()  
                    AND parts.ele.processes.reset.isGood() 
                    AND parts.roc.processes.reset.isGood() 
                    AND parts.ron.processes.reset.isGood() 
                    //AND parts.fwAxis.processes.reset.isGood() 
                THEN
                    processes.reset._state := 10;
                ELSE
                    processes.reset.setActualStatus('Failed to reset the axes');
                    processes.reset._state := 999;
                END_IF
			END_IF  
        10:
            // just finish!
            processes.reset._state := 1000;
        999:
            // done
            processes.reset.setBad();
            processes.reset.setFinished();
        1000:
            // all done!
            processes.reset.setActualStatus('Reset done');
            processes.reset.setGood();
            processes.reset.setFinished();
	END_CASE
    
END_IF
END_METHOD

METHOD FB_init : BOOL
VAR_INPUT
	bInitRetains : BOOL; // if TRUE, the retain variables are initialized (warm start / cold start)
	bInCopyCode : BOOL;  // if TRUE, the instance afterwards gets moved into the copy code (online change)
END_VAR
parts.configManager.configure(
    editableConfigAddress       := ADR(editableConfig),
    activeConfigAddress         := ADR(config),
    configLength                := SIZEOF(editableConfig),
    editableConfigSymbolName    := GLOBAL.config.AXES_EDITABLE_CONFIG_SYMBOL_NAME,
    activeConfigSymbolName      := GLOBAL.config.AXES_ACTIVE_CONFIG_SYMBOL_NAME,
    configFilePath              := GLOBAL.config.AXES_CONFIG_FILE_PATH);
	
// put the epoch at its default value
toCppAxes.epoch := 2000.0;
END_METHOD

METHOD startTracking
VAR_INPUT
END_VAR

// do the tpoint calculations
_tpointCalculations(
    azi     := fromCppAxes.object.observedFull.az,
    ele     := fromCppAxes.object.observedFull.el,
    model   := activePointingModel,
    active  := isPointingModelActive);
    
// update the target (target is in degrees!!!)

// update the target (target is in degrees!!!)
target.updateAziEle(
        input    := fromCppAxes.object.observedFull, // radians
        deltaAzi := _tpointCalculations.deltaAzi,  // arcseconds
        deltaEle := _tpointCalculations.deltaEle); // arcseconds

// store the azi/ele/rot when starting to track
_trackingStartAzi := target.aziPos.degrees.value;
_trackingStartEle := target.elePos.degrees.value;
_trackingStartRot := target.paPos.degrees.value;

// set the shared tracking flag
isTracking := TRUE;
END_METHOD

METHOD _onFirstStart
VAR_INPUT
END_VAR
CASE _onFirstStartCurrentAction OF
    0:
        // start loading the config from XML file
        parts.configManager.processes.load.start(parts.configManager.processes.load.set.filePath);
        _onFirstStartCurrentAction := 1;
    1:
        // wait until the config has been loaded
        IF parts.configManager.processes.load.statuses.busyStatus.idle THEN
            IF parts.configManager.processes.load.statuses.healthStatus.good THEN
                _onFirstStartCurrentAction := 2;
            ELSE
                _onFirstStartCurrentAction := 999;
            END_IF
        END_IF
    2:
        // now start activating the config
        parts.configManager.processes.activate.start();
        _onFirstStartCurrentAction := 3;
    3:
        // wait until the config has been activated
        IF parts.configManager.processes.activate.statuses.busyStatus.idle THEN
            IF parts.configManager.processes.activate.statuses.healthStatus.good THEN
                _onFirstStartCurrentAction := 4;
            ELSE
                _onFirstStartCurrentAction := 999;
            END_IF
        END_IF
    4:
        // set the internal pointers
        parts.io.parts.aziDrive.parts.channelA.setInternalAxisRef(pointerToAxisRef := ADR(parts.azi.parts.physicalAxis.axis_ref));
        parts.io.parts.aziDrive.parts.channelB.setInternalAxisRef(pointerToAxisRef := ADR(parts.roc.parts.physicalAxis.axis_ref));
        parts.io.parts.ablDrive.parts.channelA.setInternalAxisRef(pointerToAxisRef := ADR(parts.azi.parts.ablAxis.axis_ref));
        parts.io.parts.ablDrive.parts.channelB.setInternalAxisRef(pointerToAxisRef := ADR(parts.ron.parts.physicalAxis.axis_ref));
        parts.io.parts.eleDrive.parts.channelA.setInternalAxisRef(pointerToAxisRef := ADR(parts.ele.parts.physicalAxis.axis_ref));
        //parts.eleDrive.parts.channelB.setInternalAxisRef(pointerToAxisRef := ADR(parts.fwAxis.parts.physicalAxis.axis_ref)); // TODO: uncomment
        
        _onFirstStartCurrentAction := 5;
    5:
        // nothing to do, done!
        ;
    999:
        // error, but nothing we can do about it now!
        ;

END_CASE
END_METHOD

METHOD _stop
VAR_INPUT
END_VAR
IF processes.stop.isBusy() THEN
    
    IF NOT processes.stop.isStarted() THEN
        processes.stop.state := 0;
        processes.stop.setStarted();
	END_IF
    
    CASE processes.stop.state OF
        0:
            processes.stop.setActualStatus('Now stopping'); 
            
            stopTracking();
            
            IF parts.azi.statuses.poweredStatus.enabled THEN
                parts.azi.processes.stop.start();
			END_IF
            IF parts.ele.statuses.poweredStatus.enabled THEN
                parts.ele.processes.stop.start();
			END_IF
            IF parts.roc.statuses.poweredStatus.enabled THEN
                parts.roc.processes.stop.start();
			END_IF
            IF parts.ron.statuses.poweredStatus.enabled THEN
                parts.ron.processes.stop.start();
			END_IF
            processes.stop.state := 1;
        1:
            IF     (parts.azi.processes.stop.isIdle() OR parts.azi.statuses.poweredStatus.disabled)
               AND (parts.ele.processes.stop.isIdle() OR parts.ele.statuses.poweredStatus.disabled)
               AND (parts.roc.processes.stop.isIdle() OR parts.roc.statuses.poweredStatus.disabled)
               AND (parts.ron.processes.stop.isIdle() OR parts.ron.statuses.poweredStatus.disabled)
            THEN
                   
                IF     (parts.azi.processes.stop.isGood() OR parts.azi.statuses.poweredStatus.disabled)
                   AND (parts.ele.processes.stop.isGood() OR parts.ele.statuses.poweredStatus.disabled)
                   AND (parts.roc.processes.stop.isGood() OR parts.roc.statuses.poweredStatus.disabled)
                   AND (parts.ron.processes.stop.isGood() OR parts.ron.statuses.poweredStatus.disabled)
                THEN
                    processes.stop.state := 1000;
                ELSE
                    processes.stop.setActualStatus('One or more axes failed');
                    processes.stop.state := 999;
                END_IF
			END_IF
        999:
            // error!
            processes.stop.setBad();
            processes.stop.setFinished();
        1000:
            // ok done
            processes.stop.setFinished();
            processes.stop.setGood();
            processes.stop.setActualStatus('Stopped');
            
		
		
    END_CASE
    
END_IF
END_METHOD

METHOD _setTarget
VAR_INPUT
END_VAR
VAR
    alphaDeg : LREAL;
    deltaDeg : LREAL;
    muAlphaDegPerYear : LREAL;
    muDeltaDegPerYear : LREAL;
END_VAR
IF processes.setTarget.isBusy() THEN
    
    IF NOT processes.setTarget.isStarted() THEN
        
        processes.setTarget._state := 0;
        processes.setTarget.setActualStatus('Setting new target');
        processes.setTarget.setStarted();
        
	END_IF
    
    CASE processes.setTarget._state OF
        0:
            // convert the input arguments into one units
            alphaDeg := AxesAlphaUnitsToDeg(
                    units := processes.setTarget.get.alphaUnits,
                    value := processes.setTarget.get.alpha);
            deltaDeg := AxesDeltaUnitsToDeg(
                    units := processes.setTarget.get.deltaUnits,
                    value := processes.setTarget.get.delta); 
            muAlphaDegPerYear := AxesMuUnitsToDegPerYear(
                    units := processes.setTarget.get.muUnits,
                    value := processes.setTarget.get.muAlpha);
            muDeltaDegPerYear := AxesMuUnitsToDegPerYear(
                    units := processes.setTarget.get.muUnits,
                    value := processes.setTarget.get.muDelta);
            
                                           
            // copy the values to the C++ task
            toCppAxes.object.rc := DEG_TO_RAD(alphaDeg);
            toCppAxes.object.dc := DEG_TO_RAD(deltaDeg);
            toCppAxes.object.pr := DEG_TO_RAD(muAlphaDegPerYear);
            toCppAxes.object.pd := DEG_TO_RAD(muDeltaDegPerYear);
            toCppAxes.object.px := processes.setTarget.get.parallax;
            toCppAxes.object.rv := processes.setTarget.get.radialVelocity;
            toCppAxes.epoch     := processes.setTarget.get.epoch;
            
            // copy the values to the target struct
            target.alpha(newDegreesValue := alphaDeg);
            target.delta(newDegreesValue := deltaDeg);
            target.muAlpha := DEG_TO_ARCSEC(muAlphaDegPerYear);
            target.muDelta := DEG_TO_ARCSEC(muDeltaDegPerYear);
            target.parallax := processes.setTarget.get.parallax;
            target.radialVelocity := processes.setTarget.get.radialVelocity;
            target.epoch := processes.setTarget.get.epoch;
            
            // store the original alpha/delta
            target.alphaStart(newDegreesValue := alphaDeg);
            target.deltaStart(newDegreesValue := deltaDeg);
            
            // reset the travelled alpha/delta due to the alpha/delta velocity
            target.alphaTravelled(newDegreesValue := 0.0);
            target.deltaTravelled(newDegreesValue := 0.0);
            
            // reset the offsets
            target.alphaOffsetted(newDegreesValue := 0.0);
            target.deltaOffsetted(newDegreesValue := 0.0);
            
            // reset the alpha/delta velocity
            target.alphaVelocity(newDegreesPerSecondValue := 0.0);
            target.deltaVelocity(newDegreesPerSecondValue := 0.0);
            
            // now we meed to wait for the C++ task to process the new target
            _setTargetTon(IN := FALSE);
            _setTargetTon(IN := TRUE, PT := GLOBAL.config.SLALIB_TASK_TIME + 2*GLOBAL.config.PLC_FAST_TASK_TIME);
            processes.setTarget._state := 1;
        1:
            processes.setTarget.setActualStatus('Waiting until the target is set');
            _setTargetTon(IN := TRUE);
            
            IF _setTargetTon.Q THEN
                IF fromCppAxes.error = TmcAxesErrors.AXES_NO_ERROR THEN
                    processes.setTarget.setActualStatus('Taget was set');
                    processes.setTarget._state := 1000;
                ELSE
                    processes.setTarget._state := 999;
                    processes.setTarget.setActualStatus(TmcAxesErrorsToString(fromCppAxes.error));
			    END_IF
			END_IF
        999:
            processes.setTarget.setFinished();
            processes.setTarget.setBad();
        1000:
            processes.setTarget.setFinished();
            processes.setTarget.setGood();
    
    
	END_CASE
    
END_IF
END_METHOD

METHOD _unlocking
VAR_INPUT
END_VAR
IF processes.unlock.statuses.busyStatus.busy THEN
	statuses.initializationStatus(state := InitializationStates.INITIALIZED);
	
	// done
	processes.unlock.setGood();
	processes.unlock.setFinished();
END_IF
END_METHOD

METHOD _stoMonitoring : RequestResults
VAR_INPUT
END_VAR
_aziStoMonitoringEdgeDetection(CLK := motionBlocking.telescopeAzimuthReleaseOK);
_eleStoMonitoringEdgeDetection(CLK := motionBlocking.telescopeElevationReleaseOK);
_rocStoMonitoringEdgeDetection(CLK := motionBlocking.telescopeRotationReleaseOK);
_ronStoMonitoringEdgeDetection(CLK := motionBlocking.telescopeRotationReleaseOK);

IF _aziStoMonitoringEdgeDetection.Q THEN
    _aziStoCounter := _aziStoCounter + 1;
    parts.azi.processes.quickStop.start();
    stopTracking();
END_IF

IF _eleStoMonitoringEdgeDetection.Q THEN
    _eleStoCounter := _eleStoCounter + 1;
    parts.ele.processes.quickStop.start();
    stopTracking();
END_IF

IF _rocStoMonitoringEdgeDetection.Q THEN
    _rocStoCounter := _rocStoCounter + 1;
    parts.roc.processes.quickStop.start();
    stopTracking();
END_IF

IF _ronStoMonitoringEdgeDetection.Q THEN
    _ronStoCounter := _ronStoCounter + 1;
    parts.ron.processes.quickStop.start();
    stopTracking();
END_IF
END_METHOD

METHOD _update_activePointingModel : RequestResults
VAR_INPUT
END_VAR
IF isPointingModelActive THEN
    CASE activePointingModelNumber OF
        0:
            activePointingModel := parts.tpoint.parts.model0.config;
        1:
            activePointingModel := parts.tpoint.parts.model1.config;
        2:
            activePointingModel := parts.tpoint.parts.model2.config;
        3:
            activePointingModel := parts.tpoint.parts.model3.config;
        4:
            activePointingModel := parts.tpoint.parts.model4.config;
        5:
            activePointingModel := parts.tpoint.parts.model5.config;
        6:
            activePointingModel := parts.tpoint.parts.model6.config;
        7:
            activePointingModel := parts.tpoint.parts.model7.config;
        8:
            activePointingModel := parts.tpoint.parts.model8.config;
        9:
            activePointingModel := parts.tpoint.parts.model9.config;
    END_CASE
END_IF
END_METHOD

METHOD _quickStop
VAR_INPUT
END_VAR
IF processes.quickStop.isBusy() THEN
    
    IF NOT processes.quickStop.isStarted() THEN
        processes.quickStop.state := 0;
        processes.quickStop.setStarted();
	END_IF
    
    CASE processes.quickStop.state OF
        0:
            processes.quickStop.setActualStatus('Now quick stopping'); 
            
            stopTracking();
            
            parts.azi.processes.quickStop.start();
            parts.ele.processes.quickStop.start();
            IF parts.roc.statuses.poweredStatus.enabled THEN
                parts.roc.processes.quickStop.start();
			END_IF
            IF parts.ron.statuses.poweredStatus.enabled THEN
                parts.ron.processes.quickStop.start();
			END_IF
            processes.quickStop.state := 1;
        1:
            IF     parts.azi.processes.quickStop.isIdle()
               AND parts.ele.processes.quickStop.isIdle()
               AND (parts.roc.processes.quickStop.isIdle() OR parts.roc.statuses.poweredStatus.disabled)
               AND (parts.ron.processes.quickStop.isIdle() OR parts.ron.statuses.poweredStatus.disabled)
            THEN
                   
                IF     parts.azi.processes.quickStop.isGood()
                   AND parts.ele.processes.quickStop.isGood()
                   AND (parts.roc.processes.quickStop.isGood() OR parts.roc.statuses.poweredStatus.disabled)
                   AND (parts.ron.processes.quickStop.isGood() OR parts.ron.statuses.poweredStatus.disabled)
                THEN
                    processes.quickStop.state := 1000;
                ELSE
                    processes.quickStop.state := 999;
                END_IF
			END_IF
        999:
            // error!
            processes.quickStop.setBad();
            processes.quickStop.setFinished();
        1000:
            // ok done
            processes.quickStop.setFinished();
            processes.quickStop.setGood();
            processes.quickStop.setActualStatus('Quick stopped');
            
		
		
    END_CASE
    
END_IF
END_METHOD

METHOD _update_activeRotator : RequestResults
VAR_INPUT
END_VAR
IF isInstrumentActive THEN
    IF activeInstrument.rocActive THEN
        activeRotator := AxesRotatorActivity.ROC_ACTIVE;
    ELSIF activeInstrument.ronActive THEN
        activeRotator := AxesRotatorActivity.RON_ACTIVE;
    ELSE
        activeRotator := AxesRotatorActivity.NONE_ACTIVE;
	END_IF
END_IF
END_METHOD

METHOD stopTracking : BOOL
VAR_INPUT
END_VAR
isTracking := FALSE;
END_METHOD

METHOD _moveAbsolute
VAR_INPUT
END_VAR
VAR
    waitingStr : STRING;
    
    aziRequested : BOOL;
    eleRequested : BOOL;
    rocRequested : BOOL;
    ronRequested : BOOL;
    
END_VAR
IF processes.moveAbsolute.isBusy() THEN
    
    aziRequested := processes.moveAbsolute.get.doAzi;
    eleRequested := processes.moveAbsolute.get.doEle;
    rocRequested := processes.moveAbsolute.get.doRoc OR (processes.moveAbsolute.get.doRot AND (activeRotator = AxesRotatorActivity.ROC_ACTIVE));
    ronRequested := processes.moveAbsolute.get.doRon OR (processes.moveAbsolute.get.doRot AND (activeRotator = AxesRotatorActivity.RON_ACTIVE));
    
    
    IF NOT processes.moveAbsolute.isStarted() THEN
        
        processes.moveAbsolute.waitingForAzi := FALSE;
        processes.moveAbsolute.waitingForEle := FALSE;
        processes.moveAbsolute.waitingForRoc := FALSE;
        processes.moveAbsolute.waitingForRon := FALSE;
            
        processes.moveAbsolute.setStarted();
        processes.moveAbsolute._state := 0;
        
    END_IF
    
    CASE processes.moveAbsolute._state OF
        
        0:
            processes.moveAbsolute.setActualStatus('Stopping the telescope');
            processes.stop.start();
            processes.moveAbsolute._state := 1;
        1:
            IF processes.stop.isIdle() THEN
                IF processes.stop.isIdle() THEN
                    processes.moveAbsolute._state := 2;
                ELSE
                    processes.moveAbsolute._state := 999;
                    processes.moveAbsolute.setActualStatus('Could not stop');
				END_IF
			END_IF
        2:
            processes.moveAbsolute.setActualStatus('Moving absolute');
            
            IF aziRequested THEN
                parts.azi.processes.moveAbsolute.start(units := processes.moveAbsolute.get.units, processes.moveAbsolute.get.azi, offset := 0);
                processes.moveAbsolute.waitingForAzi := TRUE;
            END_IF
            
            IF eleRequested THEN
                parts.ele.processes.moveAbsolute.start(units := processes.moveAbsolute.get.units, processes.moveAbsolute.get.ele, offset := 0);
                processes.moveAbsolute.waitingForEle := TRUE;
            END_IF
            
            IF processes.moveAbsolute.get.doRot THEN
                // ROC has priority of RON (should never happen, but anyway...)
                IF rocRequested THEN
                    parts.roc.processes.moveAbsolute.start(units := processes.moveAbsolute.get.units, processes.moveAbsolute.get.rot, offset := 0);
                    processes.moveAbsolute.waitingForRoc := TRUE;
                END_IF
                IF ronRequested THEN
                    parts.ron.processes.moveAbsolute.start(units := processes.moveAbsolute.get.units, processes.moveAbsolute.get.rot, offset := 0);
                    processes.moveAbsolute.waitingForRon := TRUE;
                END_IF
            ELSIF processes.moveAbsolute.get.doRoc THEN
                parts.roc.processes.moveAbsolute.start(units := processes.moveAbsolute.get.units, processes.moveAbsolute.get.roc, offset := 0);
                processes.moveAbsolute.waitingForRoc := TRUE;
            ELSIF processes.moveAbsolute.get.doRon THEN
                parts.ron.processes.moveAbsolute.start(units := processes.moveAbsolute.get.units, processes.moveAbsolute.get.ron, offset := 0);
                processes.moveAbsolute.waitingForRon := TRUE;
            END_IF
            
            IF  NOT (processes.moveAbsolute.waitingForAzi OR processes.moveAbsolute.waitingForEle OR processes.moveAbsolute.waitingForRoc OR processes.moveAbsolute.waitingForRon) THEN
                processes.moveAbsolute.setActualStatus('No move requested');
                processes.moveAbsolute._state := 1000;
            ELSE
                processes.moveAbsolute._state := 3;
            END_IF
        3:
            
            IF processes.moveAbsolute.waitingForAzi THEN
                processes.moveAbsolute.waitingForAzi := parts.azi.processes.moveAbsolute.isBusy();
            END_IF
            IF processes.moveAbsolute.waitingForEle THEN
                processes.moveAbsolute.waitingForEle := parts.ele.processes.moveAbsolute.isBusy();
            END_IF
            IF processes.moveAbsolute.waitingForRoc THEN
                processes.moveAbsolute.waitingForRoc := parts.roc.processes.moveAbsolute.isBusy();
            END_IF
            IF processes.moveAbsolute.waitingForRon THEN
                processes.moveAbsolute.waitingForRon := parts.ron.processes.moveAbsolute.isBusy();
            END_IF
            
            IF processes.moveAbsolute.waitingForAzi OR processes.moveAbsolute.waitingForEle OR processes.moveAbsolute.waitingForRoc OR processes.moveAbsolute.waitingForRon THEN
                
                waitingStr := '';
                IF processes.moveAbsolute.waitingForAzi THEN
                    waitingStr := CONCAT(waitingStr, 'AZI');
                END_IF
                IF processes.moveAbsolute.waitingForEle THEN
                    IF waitingStr <> '' THEN  waitingStr := CONCAT(waitingStr, ', '); END_IF
                    waitingStr := CONCAT(waitingStr, 'ELE');
                END_IF
                IF processes.moveAbsolute.waitingForRoc THEN
                    IF waitingStr <> '' THEN  waitingStr := CONCAT(waitingStr, ', '); END_IF
                    waitingStr := CONCAT(waitingStr, 'ROC');
                END_IF
                IF processes.moveAbsolute.waitingForRon THEN
                    IF waitingStr <> '' THEN  waitingStr := CONCAT(waitingStr, ', '); END_IF
                    waitingStr := CONCAT(waitingStr, 'RON');
                END_IF
                
                processes.moveAbsolute.setActualStatus(CONCAT('Waiting for ', waitingStr));
                
            ELSE
                processes.moveAbsolute._state := 4;
            END_IF
        4:
            // update the health status
            IF      ((parts.azi.processes.moveAbsolute.isGood() OR NOT aziRequested))
                AND ((parts.ele.processes.moveAbsolute.isGood() OR NOT eleRequested))
                AND ((parts.roc.processes.moveAbsolute.isGood() OR NOT rocRequested))
                AND ((parts.ron.processes.moveAbsolute.isGood() OR NOT ronRequested)) 
            THEN
                processes.moveAbsolute.setActualStatus('Move finished');
                processes.moveAbsolute._state := 1000;
            ELSE
                processes.moveAbsolute._state := 999;
                processes.moveAbsolute.setActualStatus('One or more axes failed');
            END_IF
        999:
            processes.moveAbsolute.setFinished();
            processes.moveAbsolute.setBad();
        1000:
            processes.moveAbsolute.setFinished();
            processes.moveAbsolute.setGood();
    
	END_CASE
        

END_IF
END_METHOD

METHOD _callOnce
VAR_INPUT
END_VAR
VAR
END_VAR
// slalib returns angles within a certain range (e.g. [0..2PI]).
// During a crossing of the edges of this range (e.g. going from 2PI to 0), 
// we must continue to increase or decrease the value in order to not upset the tracking
_slalibSmoothener(
    enableSmoothening := processes.setTarget.isIdle() AND isTracking,
    fromCppAxes       := fromCppAxes);

// do the tpoint calculations
_tpointCalculations(
    azi     := fromCppAxes.object.observedFull.az,
    ele     := fromCppAxes.object.observedFull.el,
    model   := activePointingModel,
    active  := isPointingModelActive,
    aziSign := config.tpointAziSign,
    eleSign := config.tpointEleSign,
    deltaAziSign := config.tpointDeltaAziSign,
    deltaEleSign := config.tpointDeltaEleSign,
    oldFormulas := config.tpointOldFormulas);
    
// update the target (target is in degrees!!!)
target.updateAziEle(
        input    := fromCppAxes.object.observedFull, // radians
        deltaAzi := _tpointCalculations.deltaAzi,  // arcseconds
        deltaEle := _tpointCalculations.deltaEle); // arcseconds

// call the logic that must be executed just once, of the axes:
parts.azi.callOnce(
    dcTime              := timing.fromCppTiming.utc.dcTime,
    targetPosDeg        := target.aziPos.degrees.value, 
    targetVeloDegPerSec := target.aziVelo.degreesPerSecond.value, 
    targetAccDegPerSec2 := target.aziAcc.newDegreesPerSquareSecondValue, 
    trackingStart       := _trackingStartAzi, 
    isTracking          := isTracking,
    modelDelta          := ARCSEC_TO_DEG(_tpointCalculations.deltaAzi) );
    
parts.ele.callOnce(
    dcTime              := timing.fromCppTiming.utc.dcTime,
    targetPosDeg        := target.elePos.degrees.value, 
    targetVeloDegPerSec := target.eleVelo.degreesPerSecond.value, 
    targetAccDegPerSec2 := target.eleAcc.newDegreesPerSquareSecondValue, 
    trackingStart       := _trackingStartEle, 
    isTracking          := isTracking,
    modelDelta          := ARCSEC_TO_DEG(_tpointCalculations.deltaEle) );

parts.roc.callOnce(
    dcTime              := timing.fromCppTiming.utc.dcTime,
    targetPosDeg        := target.paPos.degrees.value * config.rocPositionAngleSign, 
    targetVeloDegPerSec := target.paVelo.degreesPerSecond.value * config.rocPositionAngleSign, 
    targetAccDegPerSec2 := target.paAcc.newDegreesPerSquareSecondValue,  // NOT multiply by config.rocPositionAngleSign??? because acceleration independent of direction??
    trackingStart       := _trackingStartRot * config.rocPositionAngleSign,
    isTracking          := isTracking );
parts.ron.callOnce(
    dcTime              := timing.fromCppTiming.utc.dcTime,
    targetPosDeg        := target.paPos.degrees.value * config.ronPositionAngleSign,
    targetVeloDegPerSec := target.paVelo.degreesPerSecond.value * config.ronPositionAngleSign,
    targetAccDegPerSec2 := target.paAcc.newDegreesPerSquareSecondValue, 
    trackingStart       := _trackingStartRot * config.ronPositionAngleSign,
    isTracking          := isTracking);
END_METHOD

METHOD _point
VAR_INPUT
END_VAR
VAR
    waitingStr : STRING;
END_VAR
IF processes.point.isBusy() THEN
    
    IF NOT processes.point.isStarted() THEN
        processes.point.state := 0;
        processes.point.setStarted();
        
        _pointRocRequested := parts.roc.statuses.poweredStatus.enabled OR processes.point.get.doRocOffset OR activeRotator = AxesRotatorActivity.ROC_ACTIVE;
        _pointRonRequested := parts.ron.statuses.poweredStatus.enabled OR processes.point.get.doRonOffset OR activeRotator = AxesRotatorActivity.RON_ACTIVE;
        
        IF _pointRocRequested THEN
            IF processes.point.get.doRocOffset THEN
                _pointRocOffset := processes.point.get.rocOffset;
            ELSIF processes.point.get.doRotOffset AND activeRotator = AxesRotatorActivity.ROC_ACTIVE THEN
                _pointRocOffset := processes.point.get.rotOffset;
            ELSE
                _pointRocOffset := 0.0;
			END_IF
		END_IF

        IF _pointRonRequested THEN
            IF processes.point.get.doRonOffset THEN
                _pointRonOffset := processes.point.get.ronOffset;
            ELSIF processes.point.get.doRotOffset AND activeRotator = AxesRotatorActivity.RON_ACTIVE THEN
                _pointRonOffset := processes.point.get.ronOffset;
            ELSE
                _pointRonOffset := 0.0;
			END_IF
		END_IF

	END_IF
    
    CASE processes.point.state OF
        0:
            IF    parts.azi.statuses.healthStatus.bad
               OR parts.ele.statuses.healthStatus.bad 
               OR (parts.roc.statuses.healthStatus.bad AND _pointRocRequested)
               OR (parts.ron.statuses.healthStatus.bad AND _pointRonRequested) THEN
                processes.point.state := 999;
                processes.point.setActualStatus('One or more axes in error state!');
            ELSIF statuses.poweredStatus.disabled THEN
                processes.point.state := 999;
                processes.point.setActualStatus('Power is off!');
            ELSIF    parts.azi.parts.physicalAxis.statuses.extSetGenStatus.disabled 
                  OR parts.ele.parts.physicalAxis.statuses.extSetGenStatus.disabled 
                  OR (parts.ele.parts.physicalAxis.statuses.extSetGenStatus.disabled AND _pointRocRequested)
                  OR (parts.ele.parts.physicalAxis.statuses.extSetGenStatus.disabled AND _pointRonRequested) THEN
                processes.point.state := 999;
                processes.point.setActualStatus('External setpoint generators disabled!');
            ELSE
                processes.point.state := 1;
            END_IF
        1:
            processes.point.setActualStatus('Settting new target');
            
            processes.setTarget.start(
                alphaUnits      := processes.point.get.alphaUnits, 
                deltaUnits      := processes.point.get.deltaUnits,
                alpha           := processes.point.get.alpha,
                delta           := processes.point.get.delta,
                muUnits         := processes.point.get.muUnits,
                muAlpha         := processes.point.get.muAlpha,
                muDelta         := processes.point.get.muDelta,
                parallax        := processes.point.get.parallax,
                radialVelocity  := processes.point.get.radialVelocity,
                epoch           := processes.point.get.epoch);
            
            processes.point.state := 2;
             
        2:
            IF processes.setTarget.isIdle() THEN
                IF processes.setTarget.isGood() THEN
                    startTracking();
                    processes.point.state := 3;
                ELSE
                    processes.point.state := 999;
                    processes.point.setActualStatus(CONCAT('Set target error: ', processes.setTarget.actualStatus));
			    END_IF
			END_IF
        3:
            processes.point.setActualStatus('Syncing the positions');
            parts.azi.parts.virtualAxis.processes.setPosition.start(value := parts.azi.parts.physicalAxis.axis_ref.NcToPlc.ActPos); 
            parts.ele.parts.virtualAxis.processes.setPosition.start(value := parts.ele.parts.physicalAxis.axis_ref.NcToPlc.ActPos); 
            IF _pointRocRequested THEN
                parts.roc.parts.virtualAxis.processes.setPosition.start(value := parts.roc.parts.physicalAxis.axis_ref.NcToPlc.ActPos); 
            END_IF
            IF _pointRonRequested THEN
                parts.ron.parts.virtualAxis.processes.setPosition.start(value := parts.ron.parts.physicalAxis.axis_ref.NcToPlc.ActPos); 
            END_IF
            processes.point.state := 4;
        4:
            IF       parts.azi.parts.virtualAxis.processes.setPosition.isIdle() 
                AND  parts.ele.parts.virtualAxis.processes.setPosition.isIdle()
                AND  (parts.roc.parts.virtualAxis.processes.setPosition.isIdle() OR NOT _pointRocRequested)
                AND  (parts.ron.parts.virtualAxis.processes.setPosition.isIdle() OR NOT _pointRonRequested) 
            THEN
                IF      parts.azi.parts.virtualAxis.processes.setPosition.isGood() 
                    AND parts.ele.parts.virtualAxis.processes.setPosition.isGood() 
                    AND (parts.roc.parts.virtualAxis.processes.setPosition.isGood() OR NOT _pointRocRequested)
                    AND (parts.ron.parts.virtualAxis.processes.setPosition.isGood() OR NOT _pointRonRequested) 
                THEN    
                    
                    _aziPointingMoveCalculator(
                        targetPos    := _trackingStartAzi, 
                        trackingVelo := target.aziVelo.degreesPerSecond.value,
                        minPos       := config.azi.minPositionSetpoint, 
                        maxPos       := config.azi.maxPositionSetpoint,
                        actPos       := parts.azi.actPos.degrees.value,
                        doMostTravel := TRUE);
                    _elePointingMoveCalculator(
                        targetPos    := _trackingStartEle, 
                        trackingVelo := target.eleVelo.degreesPerSecond.value,
                        minPos       := config.ele.minPositionSetpoint, 
                        maxPos       := config.ele.maxPositionSetpoint,
                        actPos       := parts.ele.actPos.degrees.value,
                        doMostTravel := TRUE);
                    IF _pointRocRequested THEN
                        _rocPointingMoveCalculator(
                            targetPos    := (_trackingStartRot + _pointRocOffset) * config.rocPositionAngleSign, 
                            trackingVelo := target.paVelo.degreesPerSecond.value  * config.rocPositionAngleSign,
                            minPos       := config.roc.minPositionSetpoint, 
                            maxPos       := config.roc.maxPositionSetpoint,
                            actPos       := parts.roc.actPos.degrees.value,
                            doMostTravel := TRUE);
                    END_IF
                    IF _pointRonRequested THEN
                        _ronPointingMoveCalculator(
                            targetPos    := (_trackingStartRot + _pointRonOffset) * config.ronPositionAngleSign, 
                            trackingVelo := target.paVelo.degreesPerSecond.value * config.ronPositionAngleSign,
                            minPos       := config.ron.minPositionSetpoint, 
                            maxPos       := config.ron.maxPositionSetpoint,
                            actPos       := parts.ron.actPos.degrees.value,
                            doMostTravel := TRUE);
                    END_IF
                    
                    IF _aziPointingMoveCalculator.outOfRange AND _elePointingMoveCalculator.outOfRange THEN
                        processes.point.state := 999;
                        processes.point.setActualStatus('Azimuth and elevation out of range!');
                    ELSIF _aziPointingMoveCalculator.outOfRange THEN
                        processes.point.state := 999;
                        processes.point.setActualStatus('Azimuth out of range!');
                    ELSIF _elePointingMoveCalculator.outOfRange THEN
                        processes.point.state := 999;
                        processes.point.setActualStatus('Elevation out of range!');
                    ELSIF _rocPointingMoveCalculator.outOfRange AND _pointRocRequested THEN
                        processes.point.state := 999;
                        processes.point.setActualStatus('Cassegrain rot. out of range!');
                    ELSIF _ronPointingMoveCalculator.outOfRange AND _pointRonRequested THEN
                        processes.point.state := 999;
                        processes.point.setActualStatus('Nasmyth rot. out of range!');
                    ELSE
                        parts.azi.processes.moveAbsolute.start(units := AxesMoveUnits.DEGREES, value := _aziPointingMoveCalculator.adjustedPos, offset := 0);
                        parts.ele.processes.moveAbsolute.start(units := AxesMoveUnits.DEGREES, value := _elePointingMoveCalculator.adjustedPos, offset := 0);
                        IF parts.roc.statuses.poweredStatus.enabled THEN
                            parts.roc.processes.moveAbsolute.start(units := AxesMoveUnits.DEGREES, value := _rocPointingMoveCalculator.adjustedPos, offset := 0);
                        END_IF
                        IF parts.ron.statuses.poweredStatus.enabled THEN
                            parts.ron.processes.moveAbsolute.start(units := AxesMoveUnits.DEGREES, value := _ronPointingMoveCalculator.adjustedPos, offset := 0);
                        END_IF
                        processes.point.state := 5;
					END_IF
                ELSE
                    processes.point.state := 999;
                    processes.point.setActualStatus('Could not set virtual azi to physical azi position');
                END_IF
            END_IF
            
        5:
            IF      parts.azi.processes.moveAbsolute.isIdle() 
                AND parts.ele.processes.moveAbsolute.isIdle() 
                AND (parts.roc.processes.moveAbsolute.isIdle() OR NOT _pointRocRequested)
                AND (parts.ron.processes.moveAbsolute.isIdle() OR NOT _pointRonRequested)
            THEN
                IF      parts.azi.processes.moveAbsolute.isGood() 
                    AND parts.ele.processes.moveAbsolute.isGood() 
                    AND (parts.roc.processes.moveAbsolute.isGood() OR NOT _pointRocRequested)
                    AND (parts.ron.processes.moveAbsolute.isGood() OR NOT _pointRonRequested)
                THEN
                    processes.point.setActualStatus('Finished moving absolute');
                    processes.point.state := 6;
                ELSE
                    processes.point.setActualStatus('Axis move error');
                    processes.point.state := 999;
				END_IF
            ELSE
                waitingStr := '';
                IF parts.azi.processes.moveAbsolute.isBusy() THEN
                    waitingStr := CONCAT(waitingStr, 'AZI');
				END_IF
                IF parts.ele.processes.moveAbsolute.isBusy() THEN
                    IF waitingStr <> '' THEN waitingStr := CONCAT(waitingStr, ', '); END_IF
                    waitingStr := CONCAT(waitingStr, 'ELE');
				END_IF
                IF parts.roc.processes.moveAbsolute.isBusy() THEN
                    IF waitingStr <> '' THEN waitingStr := CONCAT(waitingStr, ', '); END_IF
                    waitingStr := CONCAT(waitingStr, 'ROC');
				END_IF
                IF parts.ron.processes.moveAbsolute.isBusy() THEN
                    IF waitingStr <> '' THEN waitingStr := CONCAT(waitingStr, ', '); END_IF
                    waitingStr := CONCAT(waitingStr, 'RON');
				END_IF
                processes.point.setActualStatus(CONCAT('Moving ', waitingStr));
                
            END_IF
        6:
            IF NOT processes.point.get.tracking THEN
                stopTracking();
			END_IF
            
            processes.point.state := 1000;
        
        999:
            // error!
            processes.point.setBad();
            processes.point.setFinished();
            // stop all axes!
            processes.stop.start();
        1000:
            // all done!
            processes.point.setGood();
            processes.point.setFinished();
    
    
	END_CASE
        

END_IF
END_METHOD

METHOD _isAtKnownPosition : BOOL
VAR_IN_OUT
    cfg : AxesKnownPositionConfig;
END_VAR

IF (cfg.doAzi OR cfg.doEle OR cfg.doRoc OR cfg.doRon) AND  (cfg.name <> '') THEN
    _isAtKnownPosition :=  
                           ((NOT cfg.doAzi) OR ABS(cfg.azi - parts.azi.actPos.degrees.value) < config.knownPositionToleranceAzi)
                       AND ((NOT cfg.doEle) OR ABS(cfg.ele - parts.ele.actPos.degrees.value) < config.knownPositionToleranceEle)
                       AND ((NOT cfg.doRoc) OR ABS(cfg.roc - parts.roc.actPos.degrees.value) < config.knownPositionToleranceRoc)
                       AND ((NOT cfg.doRon) OR ABS(cfg.ron - parts.ron.actPos.degrees.value) < config.knownPositionToleranceRon);
ELSE
    
    _isAtKnownPosition :=  FALSE;
    
END_IF
END_METHOD

METHOD _domeAccessMonitoring
VAR_INPUT
END_VAR
_personHasEnteredMonitoringEdgeDetection(CLK := domeAccess.personHasEntered);

IF _personHasEnteredMonitoringEdgeDetection.Q THEN
    
    IF statuses.poweredStatus.enabled THEN
        isPoweredOffByPersonInDome := TRUE;
        _isPoweredOffByPersonInDome_azi := parts.azi.statuses.poweredStatus.enabled;
        _isPoweredOffByPersonInDome_ele := parts.ele.statuses.poweredStatus.enabled;
        _isPoweredOffByPersonInDome_roc := parts.roc.statuses.poweredStatus.enabled;
        _isPoweredOffByPersonInDome_ron := parts.ron.statuses.poweredStatus.enabled;
        processes.powerOff.start();
    END_IF
    

END_IF


IF      isPoweredOffByPersonInDome 
    AND motionBlocking.motionAllowed 
    AND (NOT domeAccess.personHasEntered) 
    AND processes.powerOff.isIdle()
    AND statuses.busyStatus.idle THEN
    
    isPoweredOffByPersonInDome := FALSE;
    
    processes.powerOn.start(
                azi := _isPoweredOffByPersonInDome_azi, 
                ele := _isPoweredOffByPersonInDome_ele, 
                roc := _isPoweredOffByPersonInDome_roc, 
                ron := _isPoweredOffByPersonInDome_ron, 
                fw := FALSE);

END_IF

// also reset the flag in case an attempt is made to power on or reset the telescope manually

IF processes.powerOn.isBusy() OR processes.reset.isBusy() THEN
    isPoweredOffByPersonInDome := FALSE;
END_IF
END_METHOD

METHOD _update_localConditions
VAR_INPUT
END_VAR
toCppAxes.location.tk   := CELSIUS_TO_KELVIN(config.localConditions.configuredTemperature);
toCppAxes.location.phpa := config.localConditions.configuredPressure;
toCppAxes.location.rh   := config.localConditions.configuredRelativeHumidity;
toCppAxes.location.wlfq := config.localConditions.configuredObservingWavelength;
toCppAxes.location.tlr  := config.localConditions.troposphericLapseRate;
END_METHOD

METHOD _doHoming
VAR_INPUT
END_VAR

VAR
END_VAR
IF processes.doHoming.isBusy() THEN
    
    IF NOT processes.doHoming.isStarted() THEN
        processes.doHoming.state := 0;
        processes.doHoming.setStarted();
	END_IF
    
    CASE processes.doHoming.state OF
        0:
            processes.doHoming.setActualStatus('Homing the axes');
            parts.azi.processes.doHoming.start();
            parts.ele.processes.doHoming.start();
            processes.doHoming.state := 1;
        1:
            IF      parts.azi.processes.doHoming.isIdle() 
                AND parts.ele.processes.doHoming.isIdle() THEN
                
                IF      parts.azi.processes.doHoming.isGood() 
                   AND  parts.ele.processes.doHoming.isGood() THEN
                    // ok, all axes are powered off
                    processes.doHoming.state := 1000;
                ELSE
                    processes.doHoming.setActualStatus('Could not perform homing!');
                    processes.doHoming.state := 999;
                END_IF
            END_IF
        999:
            // error!
            processes.doHoming.setBad();
            processes.doHoming.setFinished();
            // stop all axes
            processes.stop.start();
        1000:
            processes.doHoming.setActualStatus('Powered off');
            // ok done
            processes.doHoming.setFinished();
            processes.doHoming.setGood();
		
    END_CASE
    
END_IF
END_METHOD

METHOD _moveRelative
VAR_INPUT
END_VAR
VAR
    waitingStr : STRING;
    aziIsGood : BOOL;
    eleIsGood : BOOL;
    rocIsGood : BOOL;
    ronIsGood : BOOL;
    
    aziRequested : BOOL;
    eleRequested : BOOL;
    rocRequested : BOOL;
    ronRequested : BOOL;
    
END_VAR
IF processes.moveRelative.isBusy() THEN
    
    aziRequested := processes.moveRelative.get.doAzi;
    eleRequested := processes.moveRelative.get.doEle;
    rocRequested := processes.moveRelative.get.doRoc OR (processes.moveRelative.get.doRot AND (activeRotator = AxesRotatorActivity.ROC_ACTIVE));
    ronRequested := processes.moveRelative.get.doRon OR (processes.moveRelative.get.doRot AND (activeRotator = AxesRotatorActivity.RON_ACTIVE));
        
    IF NOT processes.moveRelative.isStarted() THEN
        
        processes.moveRelative.setStarted();
    
        processes.moveRelative.setActualStatus('Moving relative');
        
        processes.moveRelative.waitingForAzi := FALSE;
        processes.moveRelative.waitingForEle := FALSE;
        processes.moveRelative.waitingForRoc := FALSE;
        processes.moveRelative.waitingForRon := FALSE;
        
        
        IF aziRequested THEN
            _aziMoveRelativeCalculator(
                    distance     := AxesMoveUnitsToDeg(units := processes.moveRelative.get.units, value := processes.moveRelative.get.azi), 
                    trackingVelo := target.aziVelo.degreesPerSecond.value,
                    minPos       := config.azi.minPositionSetpoint, 
                    maxPos       := config.azi.maxPositionSetpoint,
                    actPos       := parts.azi.actPos.degrees.value,
                    doMostTravel := processes.moveRelative.get.preferMostTravel);
            IF _aziMoveRelativeCalculator.outOfRange THEN
                processes.moveRelative.setActualStatus('Cannot move AZI: out of range');
                processes.moveRelative.setBad();
                processes.moveRelative.waitingForAzi := FALSE;
            ELSE
                parts.azi.processes.moveRelative.start(units := AxesMoveUnits.DEGREES, _aziMoveRelativeCalculator.adjustedDistance);
                processes.moveRelative.waitingForAzi := TRUE;
			END_IF
        END_IF
        
        IF eleRequested THEN
            _eleMoveRelativeCalculator(
                    distance     := AxesMoveUnitsToDeg(units := processes.moveRelative.get.units, value := processes.moveRelative.get.ele), 
                    trackingVelo := target.eleVelo.degreesPerSecond.value,
                    minPos       := config.ele.minPositionSetpoint, 
                    maxPos       := config.ele.maxPositionSetpoint,
                    actPos       := parts.ele.actPos.degrees.value,
                    doMostTravel := processes.moveRelative.get.preferMostTravel);
            IF _eleMoveRelativeCalculator.outOfRange THEN
                processes.moveRelative.setActualStatus('Cannot move ELE: out of range');
                processes.moveRelative.setFinished();
                processes.moveRelative.waitingForEle := FALSE;
            ELSE
                parts.ele.processes.moveRelative.start(units := AxesMoveUnits.DEGREES, _eleMoveRelativeCalculator.adjustedDistance);
                processes.moveRelative.waitingForEle := TRUE;
			END_IF
        END_IF
        
        IF processes.moveRelative.get.doRot THEN
            IF rocRequested THEN
                _rocMoveRelativeCalculator(
                        distance     := AxesMoveUnitsToDeg(units := processes.moveRelative.get.units, processes.moveRelative.get.rot), 
                        trackingVelo := target.paVelo.degreesPerSecond.value,
                        minPos       := config.roc.minPositionSetpoint, 
                        maxPos       := config.roc.maxPositionSetpoint,
                        actPos       := parts.roc.actPos.degrees.value,
                        doMostTravel := processes.moveRelative.get.preferMostTravel);
                IF _rocMoveRelativeCalculator.outOfRange THEN
                    processes.moveRelative.setActualStatus('Cannot move ROC: out of range');
                    processes.moveRelative.setFinished();
                    processes.moveRelative.waitingForRoc := FALSE;
                ELSE
                    parts.roc.processes.moveRelative.start(units := AxesMoveUnits.DEGREES, _rocMoveRelativeCalculator.adjustedDistance);
                    processes.moveRelative.waitingForRoc := TRUE;
                END_IF
            END_IF
            IF ronRequested THEN
                _ronMoveRelativeCalculator(
                        distance     := AxesMoveUnitsToDeg(units := processes.moveRelative.get.units, value := processes.moveRelative.get.rot), 
                        trackingVelo := target.paVelo.degreesPerSecond.value,
                        minPos       := config.ron.minPositionSetpoint, 
                        maxPos       := config.ron.maxPositionSetpoint,
                        actPos       := parts.ron.actPos.degrees.value,
                        doMostTravel := processes.moveRelative.get.preferMostTravel);
                IF _ronMoveRelativeCalculator.outOfRange THEN
                    processes.moveRelative.setActualStatus('Cannot move RON: out of range');
                    processes.moveRelative.setFinished();
                    processes.moveRelative.waitingForRon := FALSE;
                ELSE
                    parts.ron.processes.moveRelative.start(units := AxesMoveUnits.DEGREES, _ronMoveRelativeCalculator.adjustedDistance);
                    processes.moveRelative.waitingForRon := TRUE;
                END_IF
            END_IF
        ELSIF processes.moveRelative.get.doRoc THEN
            _rocMoveRelativeCalculator(
                    distance     := AxesMoveUnitsToDeg(units := processes.moveRelative.get.units, value := processes.moveRelative.get.roc), 
                    trackingVelo := target.paVelo.degreesPerSecond.value,
                    minPos       := config.roc.minPositionSetpoint, 
                    maxPos       := config.roc.maxPositionSetpoint,
                    actPos       := parts.roc.actPos.degrees.value,
                    doMostTravel := processes.moveRelative.get.preferMostTravel);
            IF _rocMoveRelativeCalculator.outOfRange THEN
                processes.moveRelative.setActualStatus('Cannot move ROC: out of range');
                processes.moveRelative.setFinished();
                processes.moveRelative.waitingForRoc := FALSE;
            ELSE
                parts.roc.processes.moveRelative.start(units := AxesMoveUnits.DEGREES, _rocMoveRelativeCalculator.adjustedDistance);
                processes.moveRelative.waitingForRoc := TRUE;
            END_IF
        ELSIF processes.moveRelative.get.doRon THEN
                _ronMoveRelativeCalculator(
                        distance     := AxesMoveUnitsToDeg(units := processes.moveRelative.get.units, value := processes.moveRelative.get.ron), 
                        trackingVelo := target.paVelo.degreesPerSecond.value,
                        minPos       := config.ron.minPositionSetpoint, 
                        maxPos       := config.ron.maxPositionSetpoint,
                        actPos       := parts.ron.actPos.degrees.value,
                        doMostTravel := processes.moveRelative.get.preferMostTravel);
                IF _ronMoveRelativeCalculator.outOfRange THEN
                    processes.moveRelative.setActualStatus('Cannot move RON: out of range');
                    processes.moveRelative.setFinished();
                    processes.moveRelative.waitingForRon := FALSE;
                ELSE
                    parts.ron.processes.moveRelative.start(units := AxesMoveUnits.DEGREES, _ronMoveRelativeCalculator.adjustedDistance);
                    processes.moveRelative.waitingForRon := TRUE;
                END_IF
        END_IF
        
        IF processes.moveRelative.isIdle() THEN
            processes.moveRelative.setFinished();
            processes.moveRelative.setBad();
        ELSIF  NOT (processes.moveRelative.waitingForAzi OR processes.moveRelative.waitingForEle OR processes.moveRelative.waitingForRoc OR processes.moveRelative.waitingForRon) THEN
            processes.moveRelative.setActualStatus('No move requested');
            processes.moveRelative.setFinished();
            processes.moveRelative.setGood();
		END_IF
        
    ELSE
        parts.azi.processes.moveRelative.statuses.healthStatus(isGood := TRUE, hasWarning := FALSE);
        
        aziIsGood := TRUE;
        eleIsGood := TRUE;
        rocIsGood := TRUE;
        ronIsGood := TRUE;
        
        IF processes.moveRelative.waitingForAzi THEN
            processes.moveRelative.waitingForAzi := parts.azi.processes.moveRelative.isBusy();
        END_IF
        IF processes.moveRelative.waitingForEle THEN
            processes.moveRelative.waitingForEle := parts.ele.processes.moveRelative.isBusy();
        END_IF
        IF processes.moveRelative.waitingForRoc THEN
            processes.moveRelative.waitingForRoc := parts.roc.processes.moveRelative.isBusy();
        END_IF
        IF processes.moveRelative.waitingForRon THEN
            processes.moveRelative.waitingForRon := parts.ron.processes.moveRelative.isBusy();
        END_IF
        
        // update the health status
        IF      ((parts.azi.processes.moveRelative.isGood() OR NOT aziRequested))
            AND ((parts.ele.processes.moveRelative.isGood() OR NOT eleRequested))
            AND ((parts.roc.processes.moveRelative.isGood() OR NOT rocRequested))
            AND ((parts.ron.processes.moveRelative.isGood() OR NOT ronRequested)) THEN
            processes.moveRelative.setGood();
        ELSE
            processes.moveRelative.setBad();
		END_IF
        
        // update the actual status and busy status
        IF processes.moveRelative.waitingForAzi OR processes.moveRelative.waitingForEle OR processes.moveRelative.waitingForRoc OR processes.moveRelative.waitingForRon THEN
            
